TYPE NetIdManagement :
STRUCT
	TargetNetId : STRING;
	FirstPeripheral : STRING;
END_STRUCT
END_TYPE

(* stored: Version 1.1.0.1, ProductVersion 3.1.4024.3
   DUT NetIdManagement: Id {0f77e00a-d9e4-4f2e-b7f1-8604e127e9c1} *)
